// SIMATIC S7-200 SMART project (STEP 7-Micro/WIN SMART), CPU ST30

ORGANIZATION_BLOCK MAIN:OB1
TITLE=Program Comments
BEGIN
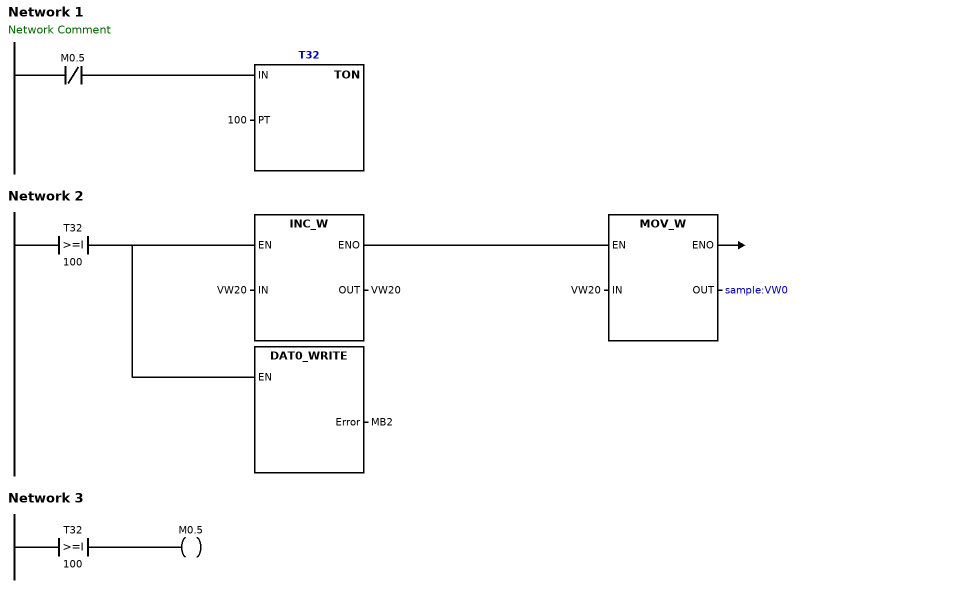
Network 1
// Network Comment
LDN    M0.5
TON    T32, 100
Network 2
LDW>=  T32, 100
LPS
INCW   VW20
AENO
MOVW   VW20, sample:VW0
LPP
CALL   DAT0_WRITE:SBR1, MB2
Network 3
LDW>=  T32, 100
=      M0.5
END_ORGANIZATION_BLOCK

// SBR1: protected block, not included

DATA_BLOCK_TAB Page_1
BEGIN
//DATA PAGE COMMENTS
//Press F1 for help and example data page
VW20     1
END_DATA_BLOCK_TAB
